// TIA Portal V17 export
// export: Created 2025-03-07T09:23:31.9832339Z, ExportSetting WithDefaults, DisplayName Totally Integrated Automation Portal, DisplayVersion V17 Update 8, DisplayName TIA Portal Openness, DisplayVersion V17 Update 8, DisplayName TIA Portal Version Control Interface, DisplayVersion V17, DisplayName SINAMICS Startdrive Advanced, DisplayVersion V17 SP2, DisplayName SINAMICS Startdrive G110M, G120, G120C, G120D, G120P, G115D, DisplayVersion V17 SP2, DisplayName SINAMICS Startdrive G130, G150, S120, S150, SINAMICS MV, S210, DisplayVersion V17 SP2, DisplayName STEP 7 Professional, DisplayVersion V17 Update 8, DisplayName SINUMERIK ONE STEP 7 Toolbox, DisplayVersion V17 Update 12, DisplayName SINUMERIK 840D sl STEP 7 Toolbox, DisplayVersion V17 Update 12, DisplayName STEP 7 Safety, DisplayVersion V17 Update 6, DisplayName WinCC Advanced, DisplayVersion V17 Update 8
ORGANIZATION_BLOCK "Cyclic interrupt"   // OB30, LAD, CyclicInterrupt
{ S7_Optimized_Access := 'TRUE' }
VERSION : 0.1
// stored: AutoNumber false, IsIECCheckEnabled false, SetENOAutomatically false
   VAR_INPUT
      Initial_Call : Bool;   // Initial call of this OB
      Event_Count : Int;   // Events discarded
   END_VAR
   VAR_TEMP
      LOOP_COUNT : Int;
   END_VAR
BEGIN

REGION Network 1: INITIALIZING OF ARRAY POINTERS FOR LOOP / Initializing of array pointers for loop
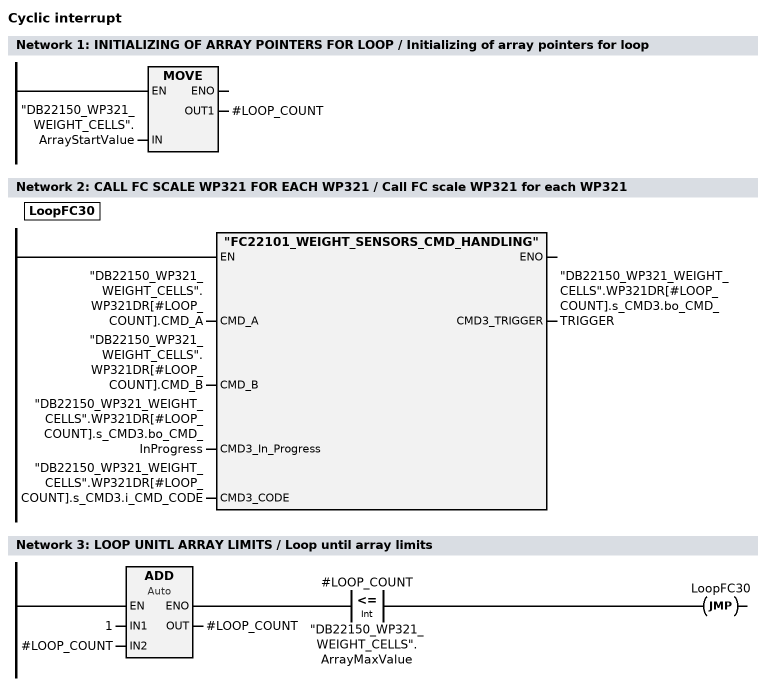
   RUNG wire#powerrail
      Move(in := "DB22150_WP321_WEIGHT_CELLS".ArrayStartValue, out1 => #LOOP_COUNT)
   END_RUNG
   // the same network as SCL:
   #LOOP_COUNT := "DB22150_WP321_WEIGHT_CELLS".ArrayStartValue;
END_REGION

REGION Network 2: CALL FC SCALE WP321 FOR EACH WP321 / Call FC scale WP321 for each WP321
   Label( LoopFC30 )
   RUNG wire#powerrail
      "FC22101_WEIGHT_SENSORS_CMD_HANDLING"(CMD_A := "DB22150_WP321_WEIGHT_CELLS".WP321DR[#LOOP_COUNT].CMD_A, CMD_B := "DB22150_WP321_WEIGHT_CELLS".WP321DR[#LOOP_COUNT].CMD_B, CMD3_In_Progress := "DB22150_WP321_WEIGHT_CELLS".WP321DR[#LOOP_COUNT].s_CMD3.bo_CMD_InProgress, CMD3_CODE := "DB22150_WP321_WEIGHT_CELLS".WP321DR[#LOOP_COUNT].s_CMD3.i_CMD_CODE, CMD3_TRIGGER => "DB22150_WP321_WEIGHT_CELLS".WP321DR[#LOOP_COUNT].s_CMD3.bo_CMD_TRIGGER)
   END_RUNG
   // the same network as SCL:
   LoopFC30:
   "FC22101_WEIGHT_SENSORS_CMD_HANDLING"(CMD_A := "DB22150_WP321_WEIGHT_CELLS".WP321DR[#LOOP_COUNT].CMD_A,
                           CMD_B := "DB22150_WP321_WEIGHT_CELLS".WP321DR[#LOOP_COUNT].CMD_B,
                           CMD3_In_Progress := "DB22150_WP321_WEIGHT_CELLS".WP321DR[#LOOP_COUNT].s_CMD3.bo_CMD_InProgress,
                           CMD3_CODE := "DB22150_WP321_WEIGHT_CELLS".WP321DR[#LOOP_COUNT].s_CMD3.i_CMD_CODE,
                           CMD3_TRIGGER => "DB22150_WP321_WEIGHT_CELLS".WP321DR[#LOOP_COUNT].s_CMD3.bo_CMD_TRIGGER);
END_REGION

REGION Network 3: LOOP UNITL ARRAY LIMITS / Loop until array limits
   RUNG wire#powerrail
      Add(in1 := 1, in2 := #LOOP_COUNT, out => #LOOP_COUNT)
      { S7_Templates := "SrcType := Int" } LE_Contact(in1 := #LOOP_COUNT, in2 := "DB22150_WP321_WEIGHT_CELLS".ArrayMaxValue)
      JumpCoil( LoopFC30 )
   END_RUNG
   // the same network as SCL:
   #LOOP_COUNT := 1 + #LOOP_COUNT;
   IF #LOOP_COUNT <= "DB22150_WP321_WEIGHT_CELLS".ArrayMaxValue THEN GOTO LoopFC30; END_IF;
END_REGION
END_ORGANIZATION_BLOCK
